TYPE NewOne :
STRUCT
END_STRUCT
END_TYPE

(* stored: Version 1.1.0.1, ProductVersion 3.1.4024.12
   DUT NewOne: Id {7b23eca7-327a-4b2e-a4ec-3021076b8163} *)
